VAR_GLOBAL CONSTANT
    
    //RAW AXES
    AXIS_1_xxx : UINT :=1;
    AXIS_2_xxx : UINT :=2;
    AXIS_3_xxx : UINT :=3;
    AXIS_4_XXX : UINT :=4;
    AXIS_HORIZONTAL_TRANSLATION : INT :=5;
    AXIS_VERTICAL_TRANSLATION_LEFT : INT :=6;
    AXIS_VERTICAL_TRANSLATION_RIGHT : INT :=7;
    AXIS_ROTATION : INT:= 8;
    
    //COMBINED MOTION AXES
    AXIS_COMBINED_VERTICAL : UINT :=9;
    
    
    
END_VAR

(* stored: Version 1.1.0.1, ProductVersion 3.1.4024.11
   GVL AXIS_NAMES: Id {7e200d6d-9582-4793-a72f-19347bc4f265} *)
